// TIA Portal V17 export
// export: Created 2021-12-03T08:13:06.2585669Z, ExportSetting WithDefaults, DisplayName Totally Integrated Automation Portal, DisplayVersion V17, DisplayName TIA Portal Openness, DisplayVersion V17, DisplayName TIA Portal Version Control Interface, DisplayVersion V17, DisplayName STEP 7 Professional, DisplayVersion V17, DisplayName STEP 7 Safety, DisplayVersion V17, DisplayName WinCC Advanced, DisplayVersion V17
DATA_BLOCK "DBI_SEW_MDX"   // DB501
AUTHOR : TSe
FAMILY : SEW_MC07
VERSION : 0.1
// stored: AutoNumber false, InstanceOfName FB_SEW_MDX, InstanceOfType FB
"FB_SEW_MDX"
   // VAR_INPUT
   //    I_AdressFrom { ExternalVisible := 'False'} : Int;
   //    I_AdressTo { ExternalVisible := 'False'} : Int;
   //    I_bForward { ExternalVisible := 'False'} : Bool;
   //    I_bBackward { ExternalVisible := 'False'} : Bool;
   //    I_bReset { ExternalVisible := 'False'} : Bool;
   //    I_bExterneFault { ExternalVisible := 'False'} : Bool;
   //    I_iReqSpeed { ExternalVisible := 'False'} : Int;
   //    I_iRampe { ExternalVisible := 'False'} : Int;
   // END_VAR
   // VAR_OUTPUT
   //    O_iFaultNumber { ExternalVisible := 'False'} : Int;
   //    O_iActSpeed { ExternalVisible := 'False'} : Int;
   //    O_iActCurrent { ExternalVisible := 'False'} : Int;
   // END_VAR
   // VAR_IN_OUT
   //    IO_bFault { ExternalVisible := 'False'} : Bool;
   // END_VAR
   // VAR RETAIN
   //    sEingangswerte { ExternalVisible := 'False'} : Struct
   //       byStatusFehlernummer { ExternalVisible := 'False'} : Byte;
   //       bStatusFreigabe { ExternalVisible := 'False'} : Bool;
   //       bStatusBetriebsbereit { ExternalVisible := 'False'} : Bool;
   //       bStatusFreigabeAusgDaten { ExternalVisible := 'False'} : Bool;
   //       bStateBit_3 { ExternalVisible := 'False'} : Bool;
   //       bStateBit_4 { ExternalVisible := 'False'} : Bool;
   //       bStatusFehler { ExternalVisible := 'False'} : Bool;
   //       bStateBit_6 { ExternalVisible := 'False'} : Bool;
   //       bStateBit_7 { ExternalVisible := 'False'} : Bool;
   //       iAktGeschwindigkeit { ExternalVisible := 'False'} : Int;
   //       iAktStrom { ExternalVisible := 'False'} : Int;
   //    END_STRUCT;
   //    sAusgangswerte { ExternalVisible := 'False'} : Struct
   //       bRichtung { ExternalVisible := 'False'} : Bool;
   //       bMotorVor { ExternalVisible := 'False'} : Bool;
   //       bMotorZurueck { ExternalVisible := 'False'} : Bool;
   //       bFestsollwert1 { ExternalVisible := 'False'} : Bool;
   //       bFestsollwert2 { ExternalVisible := 'False'} : Bool;
   //       bFestsollwertUmschaltung { ExternalVisible := 'False'} : Bool;
   //       bControlBit_14 { ExternalVisible := 'False'} : Bool;
   //       bControlBit_15 { ExternalVisible := 'False'} : Bool;
   //       bReglersperre { ExternalVisible := 'False'} : Bool;
   //       bFreigabe { ExternalVisible := 'False'} : Bool;
   //       bFreigabemitRampe { ExternalVisible := 'False'} : Bool;
   //       bControlBit_3 { ExternalVisible := 'False'} : Bool;
   //       bControlBit_4 { ExternalVisible := 'False'} : Bool;
   //       bControlBit_5 { ExternalVisible := 'False'} : Bool;
   //       bResetFehler { ExternalVisible := 'False'} : Bool;
   //       bControlBit_7 { ExternalVisible := 'False'} : Bool;
   //       iVorgabeGeschwindigkeit { ExternalVisible := 'False'} : Int;
   //       iRampe { ExternalVisible := 'False'} : Int;
   //    END_STRUCT;
   //    sSimulation { ExternalVisible := 'False'} : Struct
   //       Speed { ExternalVisible := 'False'} : Int;
   //    END_STRUCT;
   // END_VAR
BEGIN
END_DATA_BLOCK
